Staubli VAL3: duplicate.pgx

public program duplicate(string x_sCopy (dimensions=1), string x_sPaste (dimensions=1), num& x_nResult[] (dimensions=1))
  local num i
  local num l_nSize
  local string l_sItem
  local bool l_bFound
begin
  //
  // return -1 if present
  //
  // create a new one
  call new(x_sPaste,i)
  // duplicate
  saveProg:pProg[x_sPaste]=saveProg:pProg[x_sCopy]
  saveProg:pProg[x_sPaste].sID=x_sPaste
end
